{attribute 'qualified_only'}
{attribute 'strict'}
TYPE EExpressionType :
(
	none := 0,
	boolean := 1,
	comparison := 2,
	value := 3
);
END_TYPE

(* stored: Version 1.1.0.1
   DUT EExpressionType: Id {28617026-6187-454d-85c0-c71c15d16cc7} *)
